// TIA Portal project "pick and place" (V17)
// Vorlageprojekt für das Buch mit Zielsystem S7-1200

(* hardware
DEVICE "S7-1200-Station_1"  S7-1200 Station
   slot 0: "Baugruppenträger_0"  Rack  V1.0
   slot 1: "PLC_1"  CPU 1211C DC/DC/DC  6ES7 211-1AE40-0XB0  V4.1
*)

// ===== PLC "PLC_1"  CPU 1211C DC/DC/DC =====

VAR_GLOBAL   // PLC tag table "Standard-Variablentabelle"
   "item at entry" AT %I0.0 : Bool;
   "item at exit" AT %I0.1 : Bool;
   "moving x" AT %I0.2 : Bool;
   "moving z" AT %I0.3 : Bool;
   "item detected" AT %I0.4 : Bool;
   "start" AT %I0.5 : Bool;
   "reset" AT %I0.6 : Bool;
   "stop" AT %I0.7 : Bool;
   "e stop" AT %I1.0 : Bool;
   "auto" AT %I1.1 : Bool;
   "FACTORY io run" AT %I1.2 : Bool;
   "entry conv" AT %Q0.0 : Bool;
   "exit conv" AT %Q0.1 : Bool;
   "move x" AT %Q0.2 : Bool;
   "move z" AT %Q0.3 : Bool;
   "grab" AT %Q0.4 : Bool;
   "start light" AT %Q0.5 : Bool;
   "reset light" AT %Q0.6 : Bool;
   "stop light" AT %Q0.7 : Bool;
   "counter" AT %QD30 : DInt;
   "reset count" AT %M0.0 : Bool;
   "Tag_1" AT %M0.1 : Bool;
   "Tag_2" AT %M0.2 : Bool;
END_VAR

DATA_BLOCK "modes"   // DB2
{ S7_Optimized_Access := 'TRUE' }
VERSION : 0.1
   VAR
      "stop mode" : Bool;
      "start mode" : Bool;
      "auto mode" : Bool;
      "reset mode" : Bool;
      "e stop mode" : Bool;
   END_VAR
BEGIN
END_DATA_BLOCK

DATA_BLOCK "steps"   // DB4
{ S7_Optimized_Access := 'TRUE' }
VERSION : 0.1
   VAR
      "next step" : Int := 0;
      "curent step" : Int := 0;
   END_VAR
BEGIN
END_DATA_BLOCK

// folder: System blocks/Program resources

DATA_BLOCK "count"   // DB1
{ S7_Optimized_Access := 'TRUE' }
AUTHOR : Simatic
FAMILY : IEC
NAME : CNTR
VERSION : 1.0
// stored: InstanceOfName IEC_COUNTER
"IEC_COUNTER"
BEGIN
END_DATA_BLOCK

// folder: (top level)

FUNCTION "1 operation modes" : Void   // FC1, LAD
{ S7_Optimized_Access := 'TRUE' }
VERSION : 0.1
BEGIN

REGION Network 1: start mode
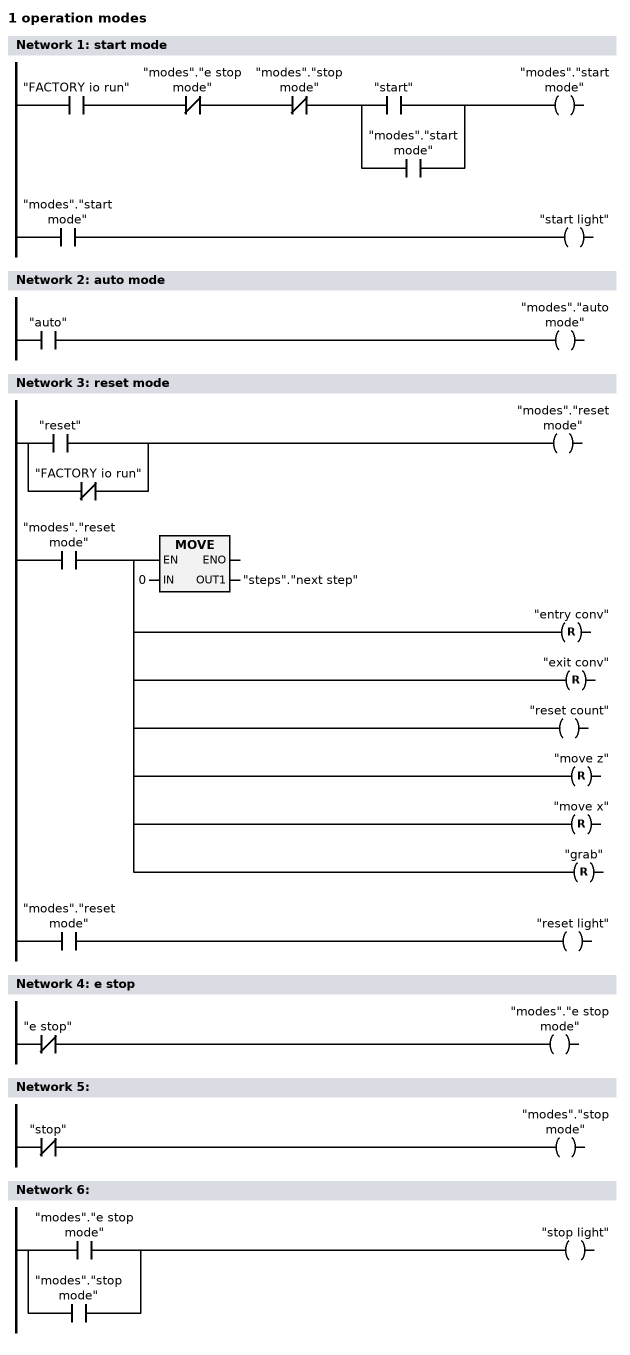
   RUNG wire#powerrail
      Contact( "FACTORY io run" )
      I_Contact( "modes"."e stop mode" )
      I_Contact( "modes"."stop mode" )
      wire#w1
      Contact( "start" )
      wire#w2
      Coil( "modes"."start mode" )
   END_RUNG
   RUNG wire#w1
      Contact( "modes"."start mode" )
   END_RUNG wire#w2
   RUNG wire#powerrail
      Contact( "modes"."start mode" )
      Coil( "start light" )
   END_RUNG
   // the same network as SCL:
   "modes"."start mode" := "FACTORY io run" AND NOT "modes"."e stop mode" AND NOT "modes"."stop mode" AND ("start" OR "modes"."start mode");
   "start light" := "modes"."start mode";
END_REGION

REGION Network 2: auto mode
   RUNG wire#powerrail
      Contact( "auto" )
      Coil( "modes"."auto mode" )
   END_RUNG
   // the same network as SCL:
   "modes"."auto mode" := "auto";
END_REGION

REGION Network 3: reset mode
   RUNG wire#powerrail
      Contact( "reset" )
      wire#w1
      Coil( "modes"."reset mode" )
   END_RUNG
   RUNG wire#powerrail
      I_Contact( "FACTORY io run" )
   END_RUNG wire#w1
   RUNG wire#powerrail
      Contact( "modes"."reset mode" )
      wire#w2
      Move(in := 0, out1 => "steps"."next step")
   END_RUNG
   RUNG wire#w2
      R_Coil( "entry conv" )
   END_RUNG
   RUNG wire#w2
      R_Coil( "exit conv" )
   END_RUNG
   RUNG wire#w2
      Coil( "reset count" )
   END_RUNG
   RUNG wire#w2
      R_Coil( "move z" )
   END_RUNG
   RUNG wire#w2
      R_Coil( "move x" )
   END_RUNG
   RUNG wire#w2
      R_Coil( "grab" )
   END_RUNG
   RUNG wire#powerrail
      Contact( "modes"."reset mode" )
      Coil( "reset light" )
   END_RUNG
   // the same network as SCL:
   "modes"."reset mode" := "reset" OR NOT "FACTORY io run";
   IF "modes"."reset mode" THEN
       "steps"."next step" := 0;
       "entry conv" := FALSE;
       "exit conv" := FALSE;
   END_IF;
   "reset count" := "modes"."reset mode";
   IF "modes"."reset mode" THEN
       "move z" := FALSE;
       "move x" := FALSE;
       "grab" := FALSE;
   END_IF;
   "reset light" := "modes"."reset mode";
END_REGION

REGION Network 4: e stop
   RUNG wire#powerrail
      I_Contact( "e stop" )
      Coil( "modes"."e stop mode" )
   END_RUNG
   // the same network as SCL:
   "modes"."e stop mode" := NOT "e stop";
END_REGION

REGION Network 5
   RUNG wire#powerrail
      I_Contact( "stop" )
      Coil( "modes"."stop mode" )
   END_RUNG
   // the same network as SCL:
   "modes"."stop mode" := NOT "stop";
END_REGION

REGION Network 6
   RUNG wire#powerrail
      Contact( "modes"."e stop mode" )
      wire#w1
      Coil( "stop light" )
   END_RUNG
   RUNG wire#powerrail
      Contact( "modes"."stop mode" )
   END_RUNG wire#w1
   // the same network as SCL:
   "stop light" := "modes"."e stop mode" OR "modes"."stop mode";
END_REGION
END_FUNCTION

FUNCTION "2 step definition" : Void   // FC2, LAD
{ S7_Optimized_Access := 'TRUE' }
VERSION : 0.1
BEGIN

REGION Network 1
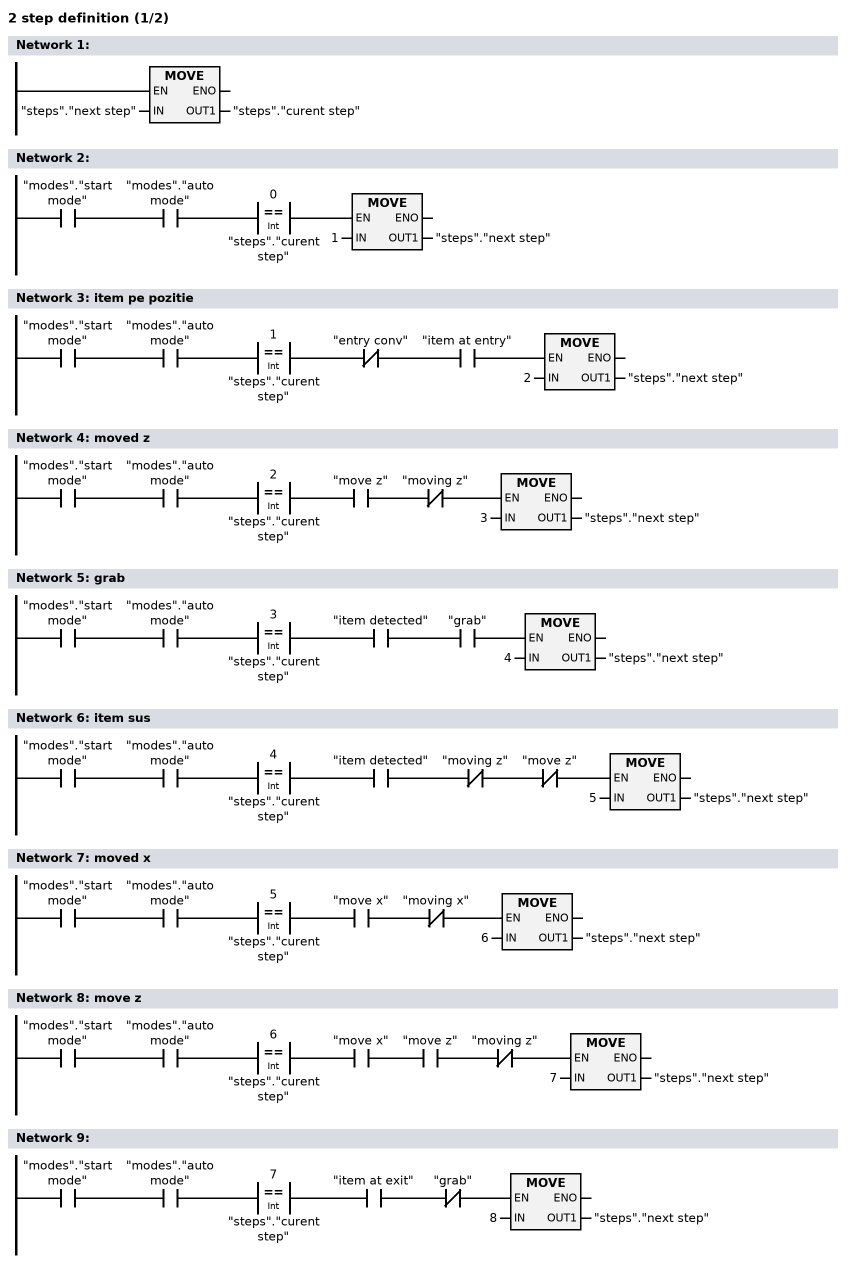
   RUNG wire#powerrail
      Move(in := "steps"."next step", out1 => "steps"."curent step")
   END_RUNG
   // the same network as SCL:
   "steps"."curent step" := "steps"."next step";
END_REGION

REGION Network 2
   RUNG wire#powerrail
      Contact( "modes"."start mode" )
      Contact( "modes"."auto mode" )
      { S7_Templates := "SrcType := Int" } EQ_Contact(in1 := 0, in2 := "steps"."curent step")
      Move(in := 1, out1 => "steps"."next step")
   END_RUNG
   // the same network as SCL:
   IF "modes"."start mode" AND "modes"."auto mode" AND (0 = "steps"."curent step") THEN
       "steps"."next step" := 1;
   END_IF;
END_REGION

REGION Network 3: item pe pozitie
   RUNG wire#powerrail
      Contact( "modes"."start mode" )
      Contact( "modes"."auto mode" )
      { S7_Templates := "SrcType := Int" } EQ_Contact(in1 := 1, in2 := "steps"."curent step")
      I_Contact( "entry conv" )
      Contact( "item at entry" )
      Move(in := 2, out1 => "steps"."next step")
   END_RUNG
   // the same network as SCL:
   IF "modes"."start mode" AND "modes"."auto mode" AND (1 = "steps"."curent step") AND NOT "entry conv" AND "item at entry" THEN
       "steps"."next step" := 2;
   END_IF;
END_REGION

REGION Network 4: moved z
   RUNG wire#powerrail
      Contact( "modes"."start mode" )
      Contact( "modes"."auto mode" )
      { S7_Templates := "SrcType := Int" } EQ_Contact(in1 := 2, in2 := "steps"."curent step")
      Contact( "move z" )
      I_Contact( "moving z" )
      Move(in := 3, out1 => "steps"."next step")
   END_RUNG
   // the same network as SCL:
   IF "modes"."start mode" AND "modes"."auto mode" AND (2 = "steps"."curent step") AND "move z" AND NOT "moving z" THEN
       "steps"."next step" := 3;
   END_IF;
END_REGION

REGION Network 5: grab
   RUNG wire#powerrail
      Contact( "modes"."start mode" )
      Contact( "modes"."auto mode" )
      { S7_Templates := "SrcType := Int" } EQ_Contact(in1 := 3, in2 := "steps"."curent step")
      Contact( "item detected" )
      Contact( "grab" )
      Move(in := 4, out1 => "steps"."next step")
   END_RUNG
   // the same network as SCL:
   IF "modes"."start mode" AND "modes"."auto mode" AND (3 = "steps"."curent step") AND "item detected" AND "grab" THEN
       "steps"."next step" := 4;
   END_IF;
END_REGION

REGION Network 6: item sus
   RUNG wire#powerrail
      Contact( "modes"."start mode" )
      Contact( "modes"."auto mode" )
      { S7_Templates := "SrcType := Int" } EQ_Contact(in1 := 4, in2 := "steps"."curent step")
      Contact( "item detected" )
      I_Contact( "moving z" )
      I_Contact( "move z" )
      Move(in := 5, out1 => "steps"."next step")
   END_RUNG
   // the same network as SCL:
   IF "modes"."start mode" AND "modes"."auto mode" AND (4 = "steps"."curent step") AND "item detected" AND NOT "moving z" AND NOT "move z" THEN
       "steps"."next step" := 5;
   END_IF;
END_REGION

REGION Network 7: moved x
   RUNG wire#powerrail
      Contact( "modes"."start mode" )
      Contact( "modes"."auto mode" )
      { S7_Templates := "SrcType := Int" } EQ_Contact(in1 := 5, in2 := "steps"."curent step")
      Contact( "move x" )
      I_Contact( "moving x" )
      Move(in := 6, out1 => "steps"."next step")
   END_RUNG
   // the same network as SCL:
   IF "modes"."start mode" AND "modes"."auto mode" AND (5 = "steps"."curent step") AND "move x" AND NOT "moving x" THEN
       "steps"."next step" := 6;
   END_IF;
END_REGION

REGION Network 8: move z
   RUNG wire#powerrail
      Contact( "modes"."start mode" )
      Contact( "modes"."auto mode" )
      { S7_Templates := "SrcType := Int" } EQ_Contact(in1 := 6, in2 := "steps"."curent step")
      Contact( "move x" )
      Contact( "move z" )
      I_Contact( "moving z" )
      Move(in := 7, out1 => "steps"."next step")
   END_RUNG
   // the same network as SCL:
   IF "modes"."start mode" AND "modes"."auto mode" AND (6 = "steps"."curent step") AND "move x" AND "move z" AND NOT "moving z" THEN
       "steps"."next step" := 7;
   END_IF;
END_REGION

REGION Network 9
   RUNG wire#powerrail
      Contact( "modes"."start mode" )
      Contact( "modes"."auto mode" )
      { S7_Templates := "SrcType := Int" } EQ_Contact(in1 := 7, in2 := "steps"."curent step")
      Contact( "item at exit" )
      I_Contact( "grab" )
      Move(in := 8, out1 => "steps"."next step")
   END_RUNG
   // the same network as SCL:
   IF "modes"."start mode" AND "modes"."auto mode" AND (7 = "steps"."curent step") AND "item at exit" AND NOT "grab" THEN
       "steps"."next step" := 8;
   END_IF;
END_REGION

REGION Network 10
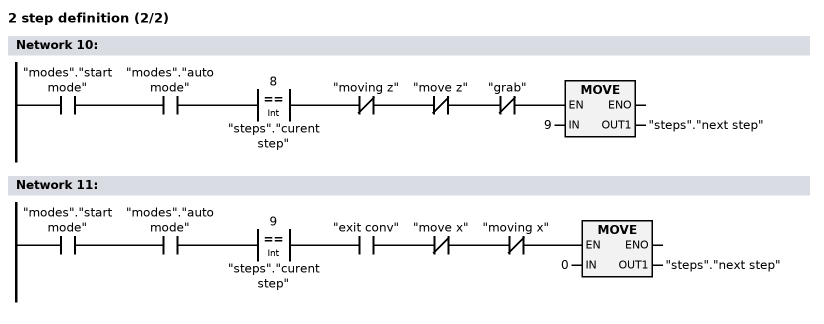
   RUNG wire#powerrail
      Contact( "modes"."start mode" )
      Contact( "modes"."auto mode" )
      { S7_Templates := "SrcType := Int" } EQ_Contact(in1 := 8, in2 := "steps"."curent step")
      I_Contact( "moving z" )
      I_Contact( "move z" )
      I_Contact( "grab" )
      Move(in := 9, out1 => "steps"."next step")
   END_RUNG
   // the same network as SCL:
   IF "modes"."start mode" AND "modes"."auto mode" AND (8 = "steps"."curent step") AND NOT "moving z" AND NOT "move z" AND NOT "grab" THEN
       "steps"."next step" := 9;
   END_IF;
END_REGION

REGION Network 11
   RUNG wire#powerrail
      Contact( "modes"."start mode" )
      Contact( "modes"."auto mode" )
      { S7_Templates := "SrcType := Int" } EQ_Contact(in1 := 9, in2 := "steps"."curent step")
      Contact( "exit conv" )
      I_Contact( "move x" )
      I_Contact( "moving x" )
      Move(in := 0, out1 => "steps"."next step")
   END_RUNG
   // the same network as SCL:
   IF "modes"."start mode" AND "modes"."auto mode" AND (9 = "steps"."curent step") AND "exit conv" AND NOT "move x" AND NOT "moving x" THEN
       "steps"."next step" := 0;
   END_IF;
END_REGION
END_FUNCTION

FUNCTION "3 step execution" : Void   // FC3, LAD
{ S7_Optimized_Access := 'TRUE' }
VERSION : 0.1
   VAR_TEMP   // added for the SCL form of the ladder/FBD networks
      _w1 : Bool;
   END_VAR
BEGIN

REGION Network 1
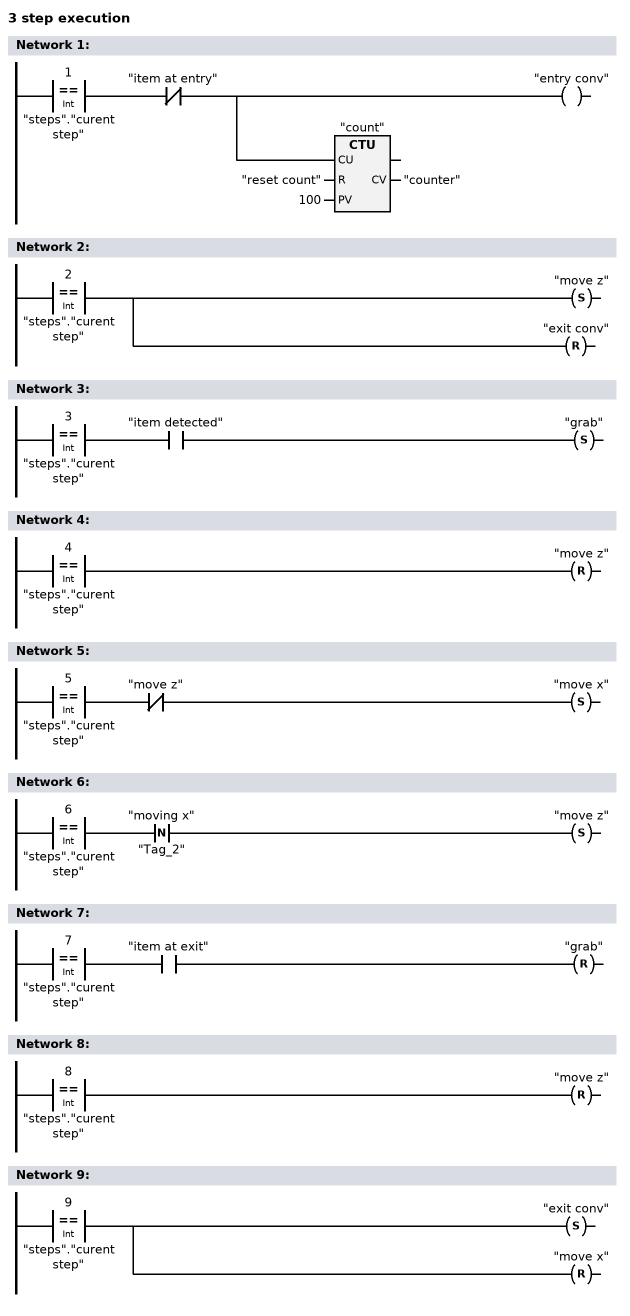
   "entry conv" := (1 = "steps"."curent step") AND NOT "item at entry";
   "count".CTU(CU := "entry conv", R := "reset count", PV := 100, CV => "counter");
END_REGION

REGION Network 2
   RUNG wire#powerrail
      { S7_Templates := "SrcType := Int" } EQ_Contact(in1 := 2, in2 := "steps"."curent step")
      wire#w1
      S_Coil( "move z" )
   END_RUNG
   RUNG wire#w1
      R_Coil( "exit conv" )
   END_RUNG
   // the same network as SCL:
   IF 2 = "steps"."curent step" THEN
       "move z" := TRUE;
       "exit conv" := FALSE;
   END_IF;
END_REGION

REGION Network 3
   RUNG wire#powerrail
      { S7_Templates := "SrcType := Int" } EQ_Contact(in1 := 3, in2 := "steps"."curent step")
      Contact( "item detected" )
      S_Coil( "grab" )
   END_RUNG
   // the same network as SCL:
   IF (3 = "steps"."curent step") AND "item detected" THEN "grab" := TRUE; END_IF;
END_REGION

REGION Network 4
   RUNG wire#powerrail
      { S7_Templates := "SrcType := Int" } EQ_Contact(in1 := 4, in2 := "steps"."curent step")
      R_Coil( "move z" )
   END_RUNG
   // the same network as SCL:
   IF 4 = "steps"."curent step" THEN "move z" := FALSE; END_IF;
END_REGION

REGION Network 5
   RUNG wire#powerrail
      { S7_Templates := "SrcType := Int" } EQ_Contact(in1 := 5, in2 := "steps"."curent step")
      I_Contact( "move z" )
      S_Coil( "move x" )
   END_RUNG
   // the same network as SCL:
   IF (5 = "steps"."curent step") AND NOT "move z" THEN "move x" := TRUE; END_IF;
END_REGION

REGION Network 6
   RUNG wire#powerrail
      { S7_Templates := "SrcType := Int" } EQ_Contact(in1 := 6, in2 := "steps"."curent step")
      N_Contact(operand := "moving x", bit := "Tag_2")
      S_Coil( "move z" )
   END_RUNG
   // the same network as SCL:
   #_w1 := (6 = "steps"."curent step") AND NOT "moving x" AND "Tag_2";   // falling edge of "moving x"
   "Tag_2" := "moving x";
   IF #_w1 THEN "move z" := TRUE; END_IF;
END_REGION

REGION Network 7
   RUNG wire#powerrail
      { S7_Templates := "SrcType := Int" } EQ_Contact(in1 := 7, in2 := "steps"."curent step")
      Contact( "item at exit" )
      R_Coil( "grab" )
   END_RUNG
   // the same network as SCL:
   IF (7 = "steps"."curent step") AND "item at exit" THEN "grab" := FALSE; END_IF;
END_REGION

REGION Network 8
   RUNG wire#powerrail
      { S7_Templates := "SrcType := Int" } EQ_Contact(in1 := 8, in2 := "steps"."curent step")
      R_Coil( "move z" )
   END_RUNG
   // the same network as SCL:
   IF 8 = "steps"."curent step" THEN "move z" := FALSE; END_IF;
END_REGION

REGION Network 9
   RUNG wire#powerrail
      { S7_Templates := "SrcType := Int" } EQ_Contact(in1 := 9, in2 := "steps"."curent step")
      wire#w1
      S_Coil( "exit conv" )
   END_RUNG
   RUNG wire#w1
      R_Coil( "move x" )
   END_RUNG
   // the same network as SCL:
   IF 9 = "steps"."curent step" THEN
       "exit conv" := TRUE;
       "move x" := FALSE;
   END_IF;
END_REGION
END_FUNCTION

FUNCTION "MHJ-PLC-Lab-Function-S71200" : Void   // FC9000, SCL
{ S7_Optimized_Access := 'TRUE' }
VERSION : 0.1
   VAR_TEMP
      rdTimeReturn : Int;
      outputTime : DTL;
      SyncVal : Byte;
      forVal : Int;
      forVal_2 : Int;
      Value : Byte;
   END_VAR
   VAR CONSTANT
      CompVal : Byte := 16#34;
      Value_01 : Byte := 16#11;
      Value_01_DW : DWord := 16#A165_D992;
      Value_02_DW : DWord := 16#58BE_4401;
   END_VAR
BEGIN

   #Value:=PEEK(area := 16#82,
        dbNumber := 0,
        byteOffset := 511);
   #Value := #Value + 1;

   POKE(area := 16#82,
        dbNumber := 0,
        byteOffset := 511,
        value := #Value);

   POKE(area:=16#81,
        dbNumber:=0,
        byteOffset:=1016,
        value:=#Value_01_DW);
   POKE(area := 16#81,
        dbNumber := 0,
        byteOffset := 1020,
        value := #Value_02_DW);

   POKE(area := 16#81,
        dbNumber := 0,
        byteOffset := 511,
        value := B#16#00);

   FOR #forVal := 0 TO 120 DO
       FOR #forVal_2:=0 TO 10 DO
           #rdTimeReturn:=RD_SYS_T(#outputTime);
           #rdTimeReturn := WR_SYS_T(#outputTime);
           #rdTimeReturn := RD_SYS_T(#outputTime);
           #rdTimeReturn := WR_SYS_T(#outputTime);
       END_FOR;
       #SyncVal:= PEEK(area := 16#81,
                      dbNumber := 0,
                      byteOffset := 511);
       IF #SyncVal = #CompVal THEN
          GOTO M_1;
       END_IF;
   END_FOR;
   RETURN;

   M_1:
   POKE(area := 16#81,
        dbNumber := 0,
        byteOffset := 511,
        value := B#16#0);
END_FUNCTION

ORGANIZATION_BLOCK "Main"   // OB1, FBD, ProgramCycle
TITLE = "Main Program Sweep (Cycle)"
{ S7_Optimized_Access := 'TRUE' }
VERSION : 0.1
   VAR_INPUT
      Initial_Call : Bool;   // Initial call of this OB
      Remanence : Bool;   // =True, if remanent data are available
   END_VAR
BEGIN

REGION Network 1: Konnektierungsbaustein für PLC-Lab
   // Im Netzwerk 1 wird der Konnektierungsbaustein für PLC-Lab aufgerufen.
   // Dieser Aufruf darf nicht entfernt werden!
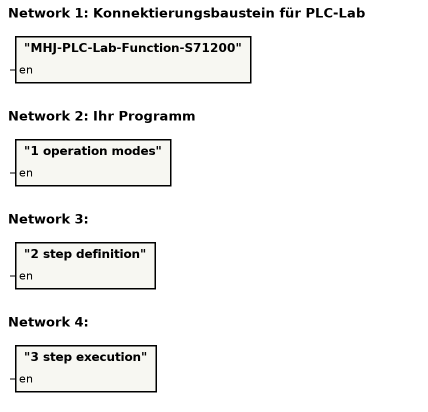
   "MHJ-PLC-Lab-Function-S71200"();
END_REGION

REGION Network 2: Ihr Programm
   // Schreiben Sie ab Netzwerk 2 Ihr Programm
   "1 operation modes"();
END_REGION

REGION Network 3
   "2 step definition"();
END_REGION

REGION Network 4
   "3 step execution"();
END_REGION
END_ORGANIZATION_BLOCK